// add command.ToolNo
CreateCommandPayload.AddUsint(_command.ToolNo);
// add command.FrameNo
CreateCommandPayload.AddUsint(_command.FrameNo);
// add command.ConnectionMode
CreateCommandPayload.AddUsint(_command.ConnectionMode);
// add command.FixedSensor
CreateCommandPayload.AddByte(_command.FixedSensor);
// add command.SensorFrame[0]
CreateCommandPayload.AddReal(_command.SensorFrame[0]);
// add command.SensorFrame[1]
CreateCommandPayload.AddReal(_command.SensorFrame[1]);
// add command.SensorFrame[2]
CreateCommandPayload.AddReal(_command.SensorFrame[2]);
// add command.SensorFrame[3]
CreateCommandPayload.AddReal(_command.SensorFrame[3]);
// add command.SensorFrame[4]
CreateCommandPayload.AddReal(_command.SensorFrame[4]);
// add command.SensorFrame[5]
CreateCommandPayload.AddReal(_command.SensorFrame[5]);
// add command.CalibrationData
CreateCommandPayload.AddUsint(_command.CalibrationData);
// add command.CalibrationData
CreateCommandPayload.AddUInt(_command.ReferenceType);
// add command.SensorValue[0]
CreateCommandPayload.AddReal(_command.SensorValue[0]);
// add command.SensorValue[1]
CreateCommandPayload.AddReal(_command.SensorValue[1]);
// add command.SensorValue[2]
CreateCommandPayload.AddReal(_command.SensorValue[2]);
// add command.SensorValue[3]
CreateCommandPayload.AddReal(_command.SensorValue[3]);
// add command.SensorValue[4]
CreateCommandPayload.AddReal(_command.SensorValue[4]);
// add command.SensorValue[5]
CreateCommandPayload.AddReal(_command.SensorValue[5]);
// add command.TargetValue[0]
CreateCommandPayload.AddReal(_command.TargetValue[0]);
// add command.TargetValue[1]
CreateCommandPayload.AddReal(_command.TargetValue[1]);
// add command.TargetValue[2]
CreateCommandPayload.AddReal(_command.TargetValue[2]);
// add command.TargetValue[3]
CreateCommandPayload.AddReal(_command.TargetValue[3]);
// add command.TargetValue[4]
CreateCommandPayload.AddReal(_command.TargetValue[4]);
// add command.TargetValue[5]
CreateCommandPayload.AddReal(_command.TargetValue[5]);
// add command.MaxVelocity
CreateCommandPayload.AddUInt(_command.MaxVelocity);
// add command.MaxDeviation[0]
CreateCommandPayload.AddReal(_command.MaxDeviation[0]);
// add command.MaxDeviation[1]
CreateCommandPayload.AddReal(_command.MaxDeviation[1]);
// add command.MaxDeviation[2]
CreateCommandPayload.AddReal(_command.MaxDeviation[2]);
// add command.MaxDeviation[3]
CreateCommandPayload.AddReal(_command.MaxDeviation[3]);
// add command.MaxDeviation[4]
CreateCommandPayload.AddReal(_command.MaxDeviation[4]);
// add command.MaxDeviation[5]
CreateCommandPayload.AddReal(_command.MaxDeviation[5]);
// add command.ErrorReaction
CreateCommandPayload.AddUsint(_command.ErrorReaction);
// add command.ErrorReferenceType
CreateCommandPayload.AddUsint(_command.ErrorReferenceType);
// add command.ErrorVector[0]
CreateCommandPayload.AddReal(_command.ErrorVector[0]);
// add command.ErrorVector[1]
CreateCommandPayload.AddReal(_command.ErrorVector[1]);
// add command.ErrorVector[2]
CreateCommandPayload.AddReal(_command.ErrorVector[2]);
// add command.ErrorVector[3]
CreateCommandPayload.AddReal(_command.ErrorVector[3]);
// add command.ErrorVector[4]
CreateCommandPayload.AddReal(_command.ErrorVector[4]);
// add command.ErrorVector[5]
CreateCommandPayload.AddReal(_command.ErrorVector[5]);
// add command.ErrorToolNo
CreateCommandPayload.AddUsint(_command.ErrorToolNo);
// add command.ErrorFrameNo
CreateCommandPayload.AddUsint(_command.ErrorFrameNo);
// add command.CompliantAxes
CreateCommandPayload.AddByte(_command.CompliantAxes);

// Create logging
CreateCommandPayloadLog(AxesGroup := AxesGroup);
END_METHOD

METHOD INTERNAL CreateCommandPayloadLog 
VAR_IN_OUT
  /// Robot assignment of function
  AxesGroup : AxesGroup; 
END_VAR
// Create log entry for Parameter start
CreateLogMessage      ( Timestamp   := AxesGroup.InternalData.SystemTime,
                        MessageType := MessageType.CMD,
                        Severity    := Severity.DEBUG,
                        MessageCode := 0,
                        MessageText := 'Create command payload with the following parameter(s) :');

// Create log entry for ToolNo
CreateLogMessagePara1 ( Timestamp   := AxesGroup.InternalData.SystemTime,
                        MessageType := MessageType.CMD,
                        Severity    := Severity.DEBUG,
                        MessageCode := 0,
                        MessageText := 'Command.ToolNo = {1}',
                        Para1       :=  USINT_TO_STRING(_command.ToolNo));
                        
// Create log entry for FrameNo
CreateLogMessagePara1 ( Timestamp   := AxesGroup.InternalData.SystemTime,
                        MessageType := MessageType.CMD,
                        Severity    := Severity.DEBUG,
                        MessageCode := 0,
                        MessageText := 'Command.FrameNo = {1}',
                        Para1       :=  USINT_TO_STRING(_command.FrameNo));
                        
// Create log entry for ConnectionMode
CreateLogMessagePara1 ( Timestamp   := AxesGroup.InternalData.SystemTime,
                        MessageType := MessageType.CMD,
                        Severity    := Severity.DEBUG,
                        MessageCode := 0,
                        MessageText := 'Command.ConnectionMode = {1}',
                        Para1       :=  SENSOR_CONNECTION_MODE_TO_STRING(_command.ConnectionMode));

// Create log entry for FixedSensor
CreateLogMessagePara1 ( Timestamp   := AxesGroup.InternalData.SystemTime,
                        MessageType := MessageType.CMD,
                        Severity    := Severity.DEBUG,
                        MessageCode := 0,
                        MessageText := 'Command.FixedSensor = {1}',
                        Para1       :=  BYTE_TO_STRING(_command.FixedSensor));

// Create log entry for SensorFrame[0]
CreateLogMessagePara1 ( Timestamp   := AxesGroup.InternalData.SystemTime,
                        MessageType := MessageType.CMD,
                        Severity    := Severity.DEBUG,
                        MessageCode := 0,
                        MessageText := 'Command.SensorFrame[0] = {1}',
                        Para1       :=  REAL_TO_STRING(_command.SensorFrame[0]));

// Create log entry for SensorFrame[1]
CreateLogMessagePara1 ( Timestamp   := AxesGroup.InternalData.SystemTime,
                        MessageType := MessageType.CMD,
                        Severity    := Severity.DEBUG,
                        MessageCode := 0,
                        MessageText := 'Command.SensorFrame[1] = {1}',
                        Para1       :=  REAL_TO_STRING(_command.SensorFrame[1]));

// Create log entry for SensorFrame[2]
CreateLogMessagePara1 ( Timestamp   := AxesGroup.InternalData.SystemTime,
                        MessageType := MessageType.CMD,
                        Severity    := Severity.DEBUG,
                        MessageCode := 0,
                        MessageText := 'Command.SensorFrame[2] = {1}',
                        Para1       :=  REAL_TO_STRING(_command.SensorFrame[2]));

// Create log entry for SensorFrame[3]
CreateLogMessagePara1 ( Timestamp   := AxesGroup.InternalData.SystemTime,
                        MessageType := MessageType.CMD,
                        Severity    := Severity.DEBUG,
                        MessageCode := 0,
                        MessageText := 'Command.SensorFrame[3] = {1}',
                        Para1       :=  REAL_TO_STRING(_command.SensorFrame[3]));
                                                
// Create log entry for SensorFrame[4]
CreateLogMessagePara1 ( Timestamp   := AxesGroup.InternalData.SystemTime,
                        MessageType := MessageType.CMD,
                        Severity    := Severity.DEBUG,
                        MessageCode := 0,
                        MessageText := 'Command.SensorFrame[4] = {1}',
                        Para1       :=  REAL_TO_STRING(_command.SensorFrame[4]));
                                                
// Create log entry for SensorFrame[5]
CreateLogMessagePara1 ( Timestamp   := AxesGroup.InternalData.SystemTime,
                        MessageType := MessageType.CMD,
                        Severity    := Severity.DEBUG,
                        MessageCode := 0,
                        MessageText := 'Command.SensorFrame[5] = {1}',
                        Para1       :=  REAL_TO_STRING(_command.SensorFrame[5]));

// Create log entry for CalibrationData
CreateLogMessagePara1 ( Timestamp   := AxesGroup.InternalData.SystemTime,
                        MessageType := MessageType.CMD,
                        Severity    := Severity.DEBUG,
                        MessageCode := 0,
                        MessageText := 'Command.CalibrationData = {1}',
                        Para1       :=  USINT_TO_STRING(_command.CalibrationData));
                        
// Create log entry for ReferenceType
CreateLogMessagePara1 ( Timestamp   := AxesGroup.InternalData.SystemTime,
                        MessageType := MessageType.CMD,
                        Severity    := Severity.DEBUG,
                        MessageCode := 0,
                        MessageText := 'Command.ReferenceType = {1}',
                        Para1       :=  REFERENCE_TYPE_TO_STRING(_command.ReferenceType));                        
                                                
// Create log entry for SensorValue[0]
CreateLogMessagePara1 ( Timestamp   := AxesGroup.InternalData.SystemTime,
                        MessageType := MessageType.CMD,
                        Severity    := Severity.DEBUG,
                        MessageCode := 0,
                        MessageText := 'Command.SensorValue[0] = {1}',
                        Para1       :=  REAL_TO_STRING(_command.SensorValue[0]));

// Create log entry for SensorValue[1]
CreateLogMessagePara1 ( Timestamp   := AxesGroup.InternalData.SystemTime,
                        MessageType := MessageType.CMD,
                        Severity    := Severity.DEBUG,
                        MessageCode := 0,
                        MessageText := 'Command.SensorValue[1] = {1}',
                        Para1       :=  REAL_TO_STRING(_command.SensorValue[1]));

// Create log entry for SensorValue[2]
CreateLogMessagePara1 ( Timestamp   := AxesGroup.InternalData.SystemTime,
                        MessageType := MessageType.CMD,
                        Severity    := Severity.DEBUG,
                        MessageCode := 0,
                        MessageText := 'Command.SensorValue[2] = {1}',
                        Para1       :=  REAL_TO_STRING(_command.SensorValue[2]));

// Create log entry for SensorValue[3]
CreateLogMessagePara1 ( Timestamp   := AxesGroup.InternalData.SystemTime,
                        MessageType := MessageType.CMD,
                        Severity    := Severity.DEBUG,
                        MessageCode := 0,
                        MessageText := 'Command.SensorValue[3] = {1}',
                        Para1       :=  REAL_TO_STRING(_command.SensorValue[3]));
                                                
// Create log entry for SensorValue[4]
CreateLogMessagePara1 ( Timestamp   := AxesGroup.InternalData.SystemTime,
                        MessageType := MessageType.CMD,
                        Severity    := Severity.DEBUG,
                        MessageCode := 0,
                        MessageText := 'Command.SensorValue[4] = {1}',
                        Para1       :=  REAL_TO_STRING(_command.SensorValue[4]));
                                                
// Create log entry for SensorValue[5]
CreateLogMessagePara1 ( Timestamp   := AxesGroup.InternalData.SystemTime,
                        MessageType := MessageType.CMD,
                        Severity    := Severity.DEBUG,
                        MessageCode := 0,
                        MessageText := 'Command.SensorValue[5] = {1}',
                        Para1       :=  REAL_TO_STRING(_command.SensorValue[5]));
                                                
// Create log entry for TargetValue[0]
CreateLogMessagePara1 ( Timestamp   := AxesGroup.InternalData.SystemTime,
                        MessageType := MessageType.CMD,
                        Severity    := Severity.DEBUG,
                        MessageCode := 0,
                        MessageText := 'Command.TargetValue[0] = {1}',
                        Para1       :=  REAL_TO_STRING(_command.TargetValue[0]));

// Create log entry for TargetValue[1]
CreateLogMessagePara1 ( Timestamp   := AxesGroup.InternalData.SystemTime,
                        MessageType := MessageType.CMD,
                        Severity    := Severity.DEBUG,
                        MessageCode := 0,
                        MessageText := 'Command.TargetValue[1] = {1}',
                        Para1       :=  REAL_TO_STRING(_command.TargetValue[1]));

// Create log entry for TargetValue[2]
CreateLogMessagePara1 ( Timestamp   := AxesGroup.InternalData.SystemTime,
                        MessageType := MessageType.CMD,
                        Severity    := Severity.DEBUG,
                        MessageCode := 0,
                        MessageText := 'Command.TargetValue[2] = {1}',
                        Para1       :=  REAL_TO_STRING(_command.TargetValue[2]));

// Create log entry for TargetValue[3]
CreateLogMessagePara1 ( Timestamp   := AxesGroup.InternalData.SystemTime,
                        MessageType := MessageType.CMD,
                        Severity    := Severity.DEBUG,
                        MessageCode := 0,
                        MessageText := 'Command.TargetValue[3] = {1}',
                        Para1       :=  REAL_TO_STRING(_command.TargetValue[3]));
                                                
// Create log entry for TargetValue[4]
CreateLogMessagePara1 ( Timestamp   := AxesGroup.InternalData.SystemTime,
                        MessageType := MessageType.CMD,
                        Severity    := Severity.DEBUG,
                        MessageCode := 0,
                        MessageText := 'Command.TargetValue[4] = {1}',
                        Para1       :=  REAL_TO_STRING(_command.TargetValue[4]));
                                                
// Create log entry for TargetValue[5]
CreateLogMessagePara1 ( Timestamp   := AxesGroup.InternalData.SystemTime,
                        MessageType := MessageType.CMD,
                        Severity    := Severity.DEBUG,
                        MessageCode := 0,
                        MessageText := 'Command.TargetValue[5] = {1}',
                        Para1       :=  REAL_TO_STRING(_command.TargetValue[5]));
                                                
// Create log entry for MaxVelocity
CreateLogMessagePara1 ( Timestamp   := AxesGroup.InternalData.SystemTime,
                        MessageType := MessageType.CMD,
                        Severity    := Severity.DEBUG,
                        MessageCode := 0,
                        MessageText := 'Command.MaxVelocity = {1}',
                        Para1       :=  UINT_TO_STRING(_command.MaxVelocity));
                        
// Create log entry for MaxDeviation[0]
CreateLogMessagePara1 ( Timestamp   := AxesGroup.InternalData.SystemTime,
                        MessageType := MessageType.CMD,
                        Severity    := Severity.DEBUG,
                        MessageCode := 0,
                        MessageText := 'Command.MaxDeviation[0] = {1}',
                        Para1       :=  REAL_TO_STRING(_command.MaxDeviation[0]));

// Create log entry for MaxDeviation[1]
CreateLogMessagePara1 ( Timestamp   := AxesGroup.InternalData.SystemTime,
                        MessageType := MessageType.CMD,
                        Severity    := Severity.DEBUG,
                        MessageCode := 0,
                        MessageText := 'Command.MaxDeviation[1] = {1}',
                        Para1       :=  REAL_TO_STRING(_command.MaxDeviation[1]));

// Create log entry for MaxDeviation[2]
CreateLogMessagePara1 ( Timestamp   := AxesGroup.InternalData.SystemTime,
                        MessageType := MessageType.CMD,
                        Severity    := Severity.DEBUG,
                        MessageCode := 0,
                        MessageText := 'Command.MaxDeviation[2] = {1}',
                        Para1       :=  REAL_TO_STRING(_command.MaxDeviation[2]));

// Create log entry for MaxDeviation[3]
CreateLogMessagePara1 ( Timestamp   := AxesGroup.InternalData.SystemTime,
                        MessageType := MessageType.CMD,
                        Severity    := Severity.DEBUG,
                        MessageCode := 0,
                        MessageText := 'Command.MaxDeviation[3] = {1}',
                        Para1       :=  REAL_TO_STRING(_command.MaxDeviation[3]));
                                                
// Create log entry for MaxDeviation[4]
CreateLogMessagePara1 ( Timestamp   := AxesGroup.InternalData.SystemTime,
                        MessageType := MessageType.CMD,
                        Severity    := Severity.DEBUG,
                        MessageCode := 0,
                        MessageText := 'Command.MaxDeviation[4] = {1}',
                        Para1       :=  REAL_TO_STRING(_command.MaxDeviation[4]));
                                                
// Create log entry for MaxDeviation[5]
CreateLogMessagePara1 ( Timestamp   := AxesGroup.InternalData.SystemTime,
                        MessageType := MessageType.CMD,
                        Severity    := Severity.DEBUG,
                        MessageCode := 0,
                        MessageText := 'Command.MaxDeviation[5] = {1}',
                        Para1       :=  REAL_TO_STRING(_command.MaxDeviation[5]));                        
                        
// Create log entry for ErrorReaction
CreateLogMessagePara1 ( Timestamp   := AxesGroup.InternalData.SystemTime,
                        MessageType := MessageType.CMD,
                        Severity    := Severity.DEBUG,
                        MessageCode := 0,
                        MessageText := 'Command.ErrorReaction = {1}',
                        Para1       :=  ERROR_REACTION_TO_STRING(_command.ErrorReaction));    
                        
// Create log entry for ErrorReferenceType
CreateLogMessagePara1 ( Timestamp   := AxesGroup.InternalData.SystemTime,
                        MessageType := MessageType.CMD,
                        Severity    := Severity.DEBUG,
                        MessageCode := 0,
                        MessageText := 'Command.ErrorReferenceType = {1}',
                        Para1       :=  REFERENCE_TYPE_TO_STRING(_command.ErrorReferenceType));     

// Create LOG entry FOR ErrorVector[0]
CreateLogMessagePara1 ( Timestamp   := AxesGroup.InternalData.SystemTime,
                        MessageType := MessageType.CMD,
                        Severity    := Severity.DEBUG,
                        MessageCode := 0,
                        MessageText := 'Command.ErrorVector[0] = {1}',
                        Para1       :=  REAL_TO_STRING(_command.ErrorVector[0]));

// Create log entry for ErrorVector[1]
CreateLogMessagePara1 ( Timestamp   := AxesGroup.InternalData.SystemTime,
                        MessageType := MessageType.CMD,
                        Severity    := Severity.DEBUG,
                        MessageCode := 0,
                        MessageText := 'Command.ErrorVector[1] = {1}',
                        Para1       :=  REAL_TO_STRING(_command.ErrorVector[1]));

// Create log entry for ErrorVector[2]
CreateLogMessagePara1 ( Timestamp   := AxesGroup.InternalData.SystemTime,
                        MessageType := MessageType.CMD,
                        Severity    := Severity.DEBUG,
                        MessageCode := 0,
                        MessageText := 'Command.ErrorVector[2] = {1}',
                        Para1       :=  REAL_TO_STRING(_command.ErrorVector[2]));

// Create log entry for ErrorVector[3]
CreateLogMessagePara1 ( Timestamp   := AxesGroup.InternalData.SystemTime,
                        MessageType := MessageType.CMD,
                        Severity    := Severity.DEBUG,
                        MessageCode := 0,
                        MessageText := 'Command.ErrorVector[3] = {1}',
                        Para1       :=  REAL_TO_STRING(_command.ErrorVector[3]));
                                                
// Create log entry for ErrorVector[4]
CreateLogMessagePara1 ( Timestamp   := AxesGroup.InternalData.SystemTime,
                        MessageType := MessageType.CMD,
                        Severity    := Severity.DEBUG,
                        MessageCode := 0,
                        MessageText := 'Command.ErrorVector[4] = {1}',
                        Para1       :=  REAL_TO_STRING(_command.ErrorVector[4]));
                                                
// Create log entry for ErrorVector[5]
CreateLogMessagePara1 ( Timestamp   := AxesGroup.InternalData.SystemTime,
                        MessageType := MessageType.CMD,
                        Severity    := Severity.DEBUG,
                        MessageCode := 0,
                        MessageText := 'Command.ErrorVector[5] = {1}',
                        Para1       :=  REAL_TO_STRING(_command.ErrorVector[5]));  

// Create log entry for ErrorToolNo
CreateLogMessagePara1 ( Timestamp   := AxesGroup.InternalData.SystemTime,
                        MessageType := MessageType.CMD,
                        Severity    := Severity.DEBUG,
                        MessageCode := 0,
                        MessageText := 'Command.ErrorToolNo = {1}',
                        Para1       :=  USINT_TO_STRING(_command.ErrorToolNo));                                                                                        

// Create log entry for ErrorFrameNo
CreateLogMessagePara1 ( Timestamp   := AxesGroup.InternalData.SystemTime,
                        MessageType := MessageType.CMD,
                        Severity    := Severity.DEBUG,
                        MessageCode := 0,
                        MessageText := 'Command.ErrorFrameNo = {1}',
                        Para1       :=  USINT_TO_STRING(_command.ErrorFrameNo));    

// Create log entry for CompliantAxes
CreateLogMessagePara1 ( Timestamp   := AxesGroup.InternalData.SystemTime,
                        MessageType := MessageType.CMD,
                        Severity    := Severity.DEBUG,
                        MessageCode := 0,
                        MessageText := 'Command.CompliantAxes = {1}',
                        Para1       :=  BYTE_TO_STRING(_command.CompliantAxes));
END_METHOD

METHOD FB_init : BOOL
VAR_INPUT
  /// if TRUE, the retain variables are initialized (warm start / cold start)
  bInitRetains : BOOL; 
  /// if TRUE, the instance afterwards gets moved into the copy code (online change)
  bInCopyCode  : BOOL;  
END_VAR
MyType := 'MC_ForceControlFB';
END_METHOD

METHOD PROTECTED OnCall
VAR_IN_OUT
  /// Robot assignment of function
  AxesGroup : AxesGroup; 
END_VAR
// call base implementation
SUPER^.OnCall(AxesGroup := AxesGroup);

// building rising and falling edges
_enable_R( CLK := Enable);
_enable_F( CLK := Enable);

CASE _stepCmd OF
  
  00:  IF ( _enable_R.Q ) 
       THEN
         // reset the rising edge
        _enable_R();       
         // reset the falling edge
        _enable_F();     

         // Check function is supported and parameter are valid ?
         IF (( CheckFunctionSupported( AxesGroup := AxesGroup )) AND
             ( CheckParameterValid   ( AxesGroup := AxesGroup )))      
         THEN
           // set busy flag
           Busy := TRUE;
           // Reset command outputs
           SysDepMemSet(pDest := ADR(OutCmd), Value := 0, DataLen := SIZEOF(OutCmd));         
           // apply command parameter
          _parCmd := ParCmd;
           // init parameter sequence
          _command.ParSeq := 1;
           // create command data
           CommandData := CreateCommandPayload(AxesGroup := AxesGroup);
           // Add command to active command register
          _uniqueID := AxesGroup.Acyclic.ActiveCommandRegister.AddCmd( pCommandFB := ADR(THIS^ ));     
           // set timeout
           SetTimeout(PT := _timeoutCmd, rTimer := _timerCmd);
           // inc step counter
          _stepCmd := _stepCmd + 1; 
         END_IF   
       END_IF
     

  01:  // Wait for responce received
       IF ( _responseReceived )
       THEN
         // reset response received flag
        _responseReceived := FALSE;

         CASE  _response.State 
         OF
           CmdMessageState.BUFFERED    : CommandBuffered    := TRUE;
           CmdMessageState.ACTIVE      : ParameterAccepted  := TRUE;
                                         Valid              := TRUE;
           CmdMessageState.ERROR       : Error              := TRUE;
         END_CASE
         
         // Done, Aborted or Error ?
         IF (_response.State >= CmdMessageState.DONE )
         THEN
           // Update results
           OutCmd.ForceStatus.ForceControlEnabled         := _response.ForceStatus.0;
           OutCmd.ForceStatus.ForceLimitEnabled           := _response.ForceStatus.1;
           OutCmd.ForceStatus.ApplyingForce               := _response.ForceStatus.2;
           OutCmd.ForceStatus.MaxDeviationReached         := _response.ForceStatus.3;
           OutCmd.ForceStatus.SpecifiedForceTorqueReached := _response.ForceStatus.4;
           OutCmd.ForceStatus.SpecifiedForceLimitReached  := _response.ForceStatus.5;
           OutCmd.ForceStatus.Bit06                       := _response.ForceStatus.6;
           OutCmd.ForceStatus.Bit07                       := _response.ForceStatus.7;  
           // set timeout
           SetTimeout(PT := _timeoutCmd, rTimer := _timerCmd);
           // inc step counter
          _stepCmd := _stepCmd + 1;
         END_IF
 
       END_IF


  02: IF (NOT Enable)
      THEN
        Reset();
	    END_IF
ELSE
  // invalid step
  ErrorID := RobotLibraryEvents.ERR_INVALID_STEP;
END_CASE



// Reset FB
IF (( _enable_R.Q ) OR
    ( _enable_F.Q ))
THEN
 _uniqueId           := 0;
 _stepCmd            := 0;
  Valid              := FALSE;
  Busy               := FALSE;
  CommandBuffered    := FALSE;
  Error              := FALSE;
  ErrorID            := 0;
  WarningID          := 0;
  InfoID             := 0;  
END_IF
END_METHOD

METHOD INTERNAL ParseResponsePayload : DINT
VAR_INPUT
  /// Response data
  ResponseData : RobotLibraryRecvDataFB;
  /// Timestamp
  Timestamp    : SystemTime;  
END_VAR
// Table 6-720: Received CMD payload (RC to PLC) of "ForceControl"
// --------------------------
// Header
// --------------------------
// Byte 00 : USINT      - ParSeq | State     
// Byte 01 : SINT       - AlarmMessageSeverity    
// Byte 02 : UINT       - AlarmMessageCode HB
// Byte 03 :            - AlarmMessageCode LB
// --------------------------
// Datablock
// --------------------------
// Byte 04 : USINT      - ForceStatus 
// --------------------------
// call base implementation to parse the header from payload buffer
ResponseData.PayloadPtr := SUPER^.ParseResponsePayload(ResponseData := ResponseData, Timestamp := Timestamp);

// copy parsed header to response
_response.ParSeq                := _rspHeader.ParSeq;
_response.State                 := _rspHeader.State;
_response.AlarmMessageSeverity  := _rspHeader.AlarmMessageSeverity;
_response.AlarmMessageCode      := _rspHeader.AlarmMessageCode;

// Get Response.ForceStatus
_response.ForceStatus := ResponseData.GetByte();

// Create logging
ParseResponsePayloadLog(ResponseData := ResponseData, Timestamp := Timestamp);
END_METHOD

METHOD INTERNAL ParseResponsePayloadLog
VAR_INPUT
  /// Response data
  ResponseData : RobotLibraryRecvDataFB;
  /// Timestamp
  Timestamp    : SystemTime;  
END_VAR
// Create log entry for Parameter start
CreateLogMessage      ( Timestamp   := Timestamp,
                        MessageType := MessageType.CMD,
                        Severity    := Severity.DEBUG,
                        MessageCode := 0,
                        MessageText := 'Parsed the following parameter(s) from response data:');
                        
// Create log entry for ForceStatus
CreateLogMessagePara1 ( Timestamp   := Timestamp,
                        MessageType := MessageType.CMD,
                        Severity    := Severity.DEBUG,
                        MessageCode := 0,
                        MessageText := 'Response.ForceStatus = {1}',
                        Para1       :=  BYTE_TO_STRING(_response.ForceStatus));
END_METHOD

METHOD PROTECTED Reset : DINT
VAR_INPUT
END_VAR
Reset := SUPER^.Reset();

Valid              := FALSE;
Busy               := FALSE;
CommandBuffered    := FALSE;
ParameterAccepted  := FALSE;
END_METHOD

END_FUNCTION_BLOCK

// Library/POUs/ForceControl/MC_ForceLimit/MC_ForceLimitFB
/// Commands specified reaction from RA when defined force/torque detected
FUNCTION_BLOCK MC_ForceLimitFB EXTENDS RobotLibraryBaseFB
// ------------------------------------------------------------------------- 
//  SRCI Robot Library                                                
// ------------------------------------------------------------------------- 
//                                                                           
//  Object:      ForceLimitFB                                       
//  Author:      Thorsten Brach                                                
//  Date:        2024-06-01
//
//  Description:                                              
//   
//                                                                           
//  Copyright: 
//    (C) 2024 Thorsten Brach. All rights reserved                                                                                                                                            
//             Licensed under the LGPL-3.0 license.
//                                                                           
//  Disclaimer:                                                                           
//    This project is provided without any guarantee and can be used for   
//    private and commercial purposes. Any use is at the user’s 
//    own risk and responsibility.
//
// -------------------------------------------------------------------------
VAR_INPUT
  /// Set TRUE to activate force limiting
  Enable            : BOOL;
  /// Command parameter 
  ParCmd            : ForceLimitParCmd;   
END_VAR

VAR_OUTPUT
  /// TRUE, while the following outputs return valid values
  Valid             : BOOL;
  /// FB is being processed
  Busy              : BOOL;
  /// Command is transferred and confirmed by the RC
  CommandBuffered   : BOOL;
  /// Receiving of input parameter values has been acknowledged by RC
  ParameterAccepted : BOOL;
  /// Command output 
  OutCmd            : ForceLimitOutCmd;      
END_VAR


VAR
  /// internal copy of command parameter 
 _parCmd            : ForceLimitParCmd;
  /// command data to send
 _command           : ForceLimitSendData;
  /// response data received
 _response          : ForceLimitRecvData;      
  /// Rising edge for enable
 _enable_R          : R_TRIG;
  /// Falling edge for enable
 _enable_F          : F_TRIG;  
END_VAR

SUPER^(AxesGroup := AxesGroup);

METHOD PROTECTED CheckFunctionSupported : BOOL
VAR_IN_OUT
  /// Robot assignment of function
  AxesGroup : AxesGroup; 
END_VAR
CheckFunctionSupported := AxesGroup.InternalData.RCSupportedFunctions.ForceLimit;

IF ( NOT CheckFunctionSupported )
THEN
  // call base implementation for set error and create log entry
  SUPER^.CheckFunctionSupported(AxesGroup := AxesGroup);
END_IF
END_METHOD

METHOD PROTECTED CheckParameterChanged : BOOL
VAR_IN_OUT
  /// Robot assignment of function
  AxesGroup    : AxesGroup; 
END_VAR
// Check ParCmd Size is > 0, because MemCmp does not work correctly with size = 0
IF (SIZEOF(ParCmd) = 0) 
THEN 
  RETURN;
END_IF

// compare memory 
_parameterChanged := ( SysDepMemCmp(pData1 := ADR(ParCmd), pData2 := ADR(_parCmd), DataLen := SIZEOF(ParCmd)) <> RobotLibraryConstants.OK );

// check parameter valid ?
_parameterValid   := CheckParameterValid( AxesGroup := AxesGroup );

IF ((  _parameterChanged        )  AND 
    (  _parameterValid          )) OR
    (  _parameterUpdateInternal )  
THEN  
  // reset internal flag for send parameter update
 _parameterUpdateInternal := FALSE;
  // update internal copy of parameters 
 _parCmd := ParCmd;
  // inc parameter sequence
 _command.ParSeq := _command.ParSeq + 1;
  // update command data  
  CommandData := CreateCommandPayload(AxesGroup := AxesGroup); // ( Access via reference to rCommandFB in ACR )
  // notify active command register 
  AxesGroup.Acyclic.ActiveCommandRegister.NotifyParameterChanged := _uniqueID;
  // Reset parameter accepted flag
  ParameterAccepted := FALSE;  
END_IF
END_METHOD

METHOD INTERNAL CreateCommandPayload : RobotLibrarySendDataFB
VAR_IN_OUT
  /// Robot assignment of function
  AxesGroup : AxesGroup; 
END_VAR
// Table 6-727: Sent CMD payload (PLC to RC) of "ForceLimit"
// --------------------------
// Header
// --------------------------
// Byte 00 : UINT       - Type HB     
// Byte 01 :            - Type LB    
// Byte 02 : USINT      - Reserve | ExecutionMode
// Byte 03 : USINT      - ParSeq  | Priority
// --------------------------
// Datablock
// --------------------------
// Byte 004 : SINT       - EmitterID[0] 
// Byte 005 : SINT       - EmitterID[1] 
// Byte 006 : SINT       - EmitterID[2] 
// Byte 007 : SINT       - EmitterID[3]
// Byte 008 : SINT       - ListenerID
// Byte 009 : BYTE       - Reserve
// Byte 010 : USINT      - ToolNo
// Byte 011 : USINT      - FrameNo
// Byte 012 : USINT      - ConnectionMode
// Byte 013 : BOOL       - FixedSensor
// Byte 014 : REAL       - SensorFrame[0] HW HB
// Byte 015 :            - SensorFrame[0] HW LB
// Byte 016 :            - SensorFrame[0] LW HB
// Byte 017 :            - SensorFrame[0] LW LB
// Byte 018 : REAL       - SensorFrame[1] HW HB
// Byte 019 :            - SensorFrame[1] HW LB
// Byte 020 :            - SensorFrame[1] LW HB
// Byte 021 :            - SensorFrame[1] LW LB
// Byte 022 : REAL       - SensorFrame[2] HW HB
// Byte 023 :            - SensorFrame[2] HW LB
// Byte 024 :            - SensorFrame[2] LW HB
// Byte 025 :            - SensorFrame[2] LW LB
// Byte 026 : REAL       - SensorFrame[3] HW HB
// Byte 027 :            - SensorFrame[3] HW LB
// Byte 028 :            - SensorFrame[3] LW HB
// Byte 029 :            - SensorFrame[3] LW LB
// Byte 030 : REAL       - SensorFrame[4] HW HB
// Byte 031 :            - SensorFrame[4] HW LB
// Byte 032 :            - SensorFrame[4] LW HB
// Byte 033 :            - SensorFrame[4] LW LB
// Byte 034 : REAL       - SensorFrame[5] HW HB
// Byte 035 :            - SensorFrame[5] HW LB
// Byte 036 :            - SensorFrame[5] LW HB
// Byte 037 :            - SensorFrame[5] LW LB
// Byte 038 : USINT      - CalibrationData
// Byte 039 : USINT      - ReferenceType
// Byte 040 : REAL       - SensorValue[0] HW HB
// Byte 041 :            - SensorValue[0] HW LB
// Byte 042 :            - SensorValue[0] LW HB
// Byte 043 :            - SensorValue[0] LW LB
// Byte 044 : REAL       - SensorValue[1] HW HB
// Byte 045 :            - SensorValue[1] HW LB
// Byte 046 :            - SensorValue[1] LW HB
// Byte 047 :            - SensorValue[1] LW LB
// Byte 048 : REAL       - SensorValue[2] HW HB
// Byte 049 :            - SensorValue[2] HW LB
// Byte 050 :            - SensorValue[2] LW HB
// Byte 051 :            - SensorValue[2] LW LB
// Byte 052 : REAL       - SensorValue[3] HW HB
// Byte 053 :            - SensorValue[3] HW LB
// Byte 054 :            - SensorValue[3] LW HB
// Byte 055 :            - SensorValue[3] LW LB
// Byte 056 : REAL       - SensorValue[4] HW HB
// Byte 057 :            - SensorValue[4] HW LB
// Byte 058 :            - SensorValue[4] LW HB
// Byte 059 :            - SensorValue[4] LW LB
// Byte 060 : REAL       - SensorValue[5] HW HB
// Byte 061 :            - SensorValue[5] HW LB
// Byte 062 :            - SensorValue[5] LW HB
// Byte 063 :            - SensorValue[5] LW LB
// Byte 064 : REAL       - Limit[0] HW HB
// Byte 065 :            - Limit[0] HW LB
// Byte 066 :            - Limit[0] LW HB
// Byte 067 :            - Limit[0] LW LB
// Byte 068 : REAL       - Limit[1] HW HB
// Byte 069 :            - Limit[1] HW LB
// Byte 070 :            - Limit[1] LW HB
// Byte 071 :            - Limit[1] LW LB
// Byte 072 : REAL       - Limit[2] HW HB
// Byte 073 :            - Limit[2] HW LB
// Byte 074 :            - Limit[2] LW HB
// Byte 075 :            - Limit[2] LW LB
// Byte 076 : REAL       - Limit[3] HW HB
// Byte 077 :            - Limit[3] HW LB
// Byte 078 :            - Limit[3] LW HB
// Byte 079 :            - Limit[3] LW LB
// Byte 080 : REAL       - Limit[4] HW HB
// Byte 081 :            - Limit[4] HW LB
// Byte 082 :            - Limit[4] LW HB
// Byte 083 :            - Limit[4] LW LB
// Byte 084 : REAL       - Limit[5] HW HB
// Byte 085 :            - Limit[5] HW LB
// Byte 086 :            - Limit[5] LW HB
// Byte 087 :            - Limit[5] LW LB


// --------------------------
// set command parameter 
_command.CmdTyp          :=  CmdType.ForceLimit;
_command.ExecMode        :=  ExecMode;
_command.ParSeq          := _command.ParSeq;
_command.Priority        :=  Priority;
_command.EmitterID[0]    := _parCmd.EmitterID;
_command.ListenerID      :=  0; {warning 'ToDo'} 
_command.Reserve         :=  0; 
_command.ToolNo          := _parCmd.ToolNo;
_command.FrameNo         := _parCmd.FrameNo;
_command.ConnectionMode  := _parCmd.ConnectionMode;
_command.FixedSensor.0   := _parCmd.FixedSensor;
_command.SensorFrame     := _parCmd.SensorFrame;
_command.CalibrationData := _parCmd.CalibrationData;
_command.ReferenceType   := _parCmd.ReferenceType;
_command.SensorValue     := _parCmd.SensorValue;
_command.ForceLimit      := _parCmd.ForceLimit;  



// copy command data to header
_cmdHeader := _command;
// call base implementation to copy header to payload buffer
CreateCommandPayload := SUPER^.CreateCommandPayload(AxesGroup := AxesGroup);


// add command.EmitterID[0]
CreateCommandPayload.AddSint(_command.EmitterID[0]);
// add command.EmitterID[1]
CreateCommandPayload.AddSint(_command.EmitterID[1]);
// add command.EmitterID[2]
CreateCommandPayload.AddSint(_command.EmitterID[2]);
// add command.EmitterID[3]
CreateCommandPayload.AddSint(_command.EmitterID[3]);
// add command.ListenerID
CreateCommandPayload.AddSint(_command.ListenerID);
// add command.Reserve
CreateCommandPayload.AddByte(_command.Reserve);
// add command.ToolNo
CreateCommandPayload.AddUsint(_command.ToolNo);
// add command.FrameNo
CreateCommandPayload.AddUsint(_command.FrameNo);
// add command.ConnectionMode
CreateCommandPayload.AddUsint(_command.ConnectionMode);
// add command.FixedSensor
CreateCommandPayload.AddByte(_command.FixedSensor);
// add command.SensorFrame[0]
CreateCommandPayload.AddReal(_command.SensorFrame[0]);
// add command.SensorFrame[1]
CreateCommandPayload.AddReal(_command.SensorFrame[1]);
// add command.SensorFrame[2]
CreateCommandPayload.AddReal(_command.SensorFrame[2]);
// add command.SensorFrame[3]
CreateCommandPayload.AddReal(_command.SensorFrame[3]);
// add command.SensorFrame[4]
CreateCommandPayload.AddReal(_command.SensorFrame[4]);
// add command.SensorFrame[5]
CreateCommandPayload.AddReal(_command.SensorFrame[5]);
// add command.CalibrationData
CreateCommandPayload.AddUsint(_command.CalibrationData);
// add command.ReferenceType
CreateCommandPayload.AddUsint(_command.ReferenceType);
// add command.SensorValue[0]
CreateCommandPayload.AddReal(_command.SensorValue[0]);
// add command.SensorValue[1]
CreateCommandPayload.AddReal(_command.SensorValue[1]);
// add command.SensorValue[2]
CreateCommandPayload.AddReal(_command.SensorValue[2]);
// add command.SensorValue[3]
CreateCommandPayload.AddReal(_command.SensorValue[3]);
// add command.SensorValue[4]
CreateCommandPayload.AddReal(_command.SensorValue[4]);
// add command.SensorValue[5]
CreateCommandPayload.AddReal(_command.SensorValue[5]);

// add command.ForceLimit[0]
CreateCommandPayload.AddReal(_command.ForceLimit[0]);
// add command.ForceLimit[1]
CreateCommandPayload.AddReal(_command.ForceLimit[1]);
// add command.ForceLimit[2]
CreateCommandPayload.AddReal(_command.ForceLimit[2]);
// add command.ForceLimit[3]
CreateCommandPayload.AddReal(_command.ForceLimit[3]);
// add command.ForceLimit[4]
CreateCommandPayload.AddReal(_command.ForceLimit[4]);
// add command.ForceLimit[5]
CreateCommandPayload.AddReal(_command.ForceLimit[5]);

// Create logging
CreateCommandPayloadLog(AxesGroup := AxesGroup);
END_METHOD

METHOD INTERNAL CreateCommandPayloadLog 
VAR_IN_OUT
  /// Robot assignment of function
  AxesGroup : AxesGroup; 
END_VAR
VAR 
  /// internal index for loops
 _idx : DINT;
END_VAR
// Create log entry for Parameter start
CreateLogMessage      ( Timestamp   := AxesGroup.InternalData.SystemTime,
                        MessageType := MessageType.CMD,
                        Severity    := Severity.DEBUG,
                        MessageCode := 0,
                        MessageText := 'Create command payload with the following parameter(s) :');

// Create log entry for EmitterID[0]
CreateLogMessagePara1 ( Timestamp   := AxesGroup.InternalData.SystemTime,
                        MessageType := MessageType.CMD,
                        Severity    := Severity.DEBUG,
                        MessageCode := 0,
                        MessageText := 'Command.EmitterID[0] = {1}',
                        Para1       :=  SINT_TO_STRING(_command.EmitterID[0]));

// Create log entry for EmitterID[x]
FOR _idx := 0 TO 3
DO
  CreateLogMessagePara2 ( Timestamp   := AxesGroup.InternalData.SystemTime,
                          MessageType := MessageType.CMD,
                          Severity    := Severity.DEBUG,
                          MessageCode := 0,
                          MessageText := 'Command.EmitterID[{2}] = {1}',
                          Para1       :=  SINT_TO_STRING(_command.EmitterID[_idx]),
                          Para2       :=  DINT_TO_STRING(_idx));
END_FOR

// Create log entry for ListenerID
CreateLogMessagePara1 ( Timestamp   := AxesGroup.InternalData.SystemTime,
                        MessageType := MessageType.CMD,
                        Severity    := Severity.DEBUG,
                        MessageCode := 0,
                        MessageText := 'Command.ListenerID = {1}',
                        Para1       :=  SINT_TO_STRING(_command.ListenerID));
                        
// Create log entry for Reserve
CreateLogMessagePara1 ( Timestamp   := AxesGroup.InternalData.SystemTime,
                        MessageType := MessageType.CMD,
                        Severity    := Severity.DEBUG,
                        MessageCode := 0,
                        MessageText := 'Command.Reserve = {1}',
                        Para1       :=  BYTE_TO_STRING(_command.Reserve));

// Create log entry for ToolNo
CreateLogMessagePara1 ( Timestamp   := AxesGroup.InternalData.SystemTime,
                        MessageType := MessageType.CMD,
                        Severity    := Severity.DEBUG,
                        MessageCode := 0,
                        MessageText := 'Command.ToolNo = {1}',
                        Para1       :=  USINT_TO_STRING(_command.ToolNo));
                        
// Create log entry for FrameNo
CreateLogMessagePara1 ( Timestamp   := AxesGroup.InternalData.SystemTime,
                        MessageType := MessageType.CMD,
                        Severity    := Severity.DEBUG,
                        MessageCode := 0,
                        MessageText := 'Command.FrameNo = {1}',
                        Para1       :=  USINT_TO_STRING(_command.FrameNo));
                        
// Create log entry for ConnectionMode
CreateLogMessagePara1 ( Timestamp   := AxesGroup.InternalData.SystemTime,
                        MessageType := MessageType.CMD,
                        Severity    := Severity.DEBUG,
                        MessageCode := 0,
                        MessageText := 'Command.ConnectionMode = {1}',
                        Para1       :=  SENSOR_CONNECTION_MODE_TO_STRING(_command.ConnectionMode));

// Create log entry for FixedSensor
CreateLogMessagePara1 ( Timestamp   := AxesGroup.InternalData.SystemTime,
                        MessageType := MessageType.CMD,
                        Severity    := Severity.DEBUG,
                        MessageCode := 0,
                        MessageText := 'Command.FixedSensor = {1}',
                        Para1       :=  BYTE_TO_STRING(_command.FixedSensor));

// Create log entry for SensorFrame[0]
CreateLogMessagePara1 ( Timestamp   := AxesGroup.InternalData.SystemTime,
                        MessageType := MessageType.CMD,
                        Severity    := Severity.DEBUG,
                        MessageCode := 0,
                        MessageText := 'Command.SensorFrame[0] = {1}',
                        Para1       :=  REAL_TO_STRING(_command.SensorFrame[0]));

// Create log entry for SensorFrame[1]
CreateLogMessagePara1 ( Timestamp   := AxesGroup.InternalData.SystemTime,
                        MessageType := MessageType.CMD,
                        Severity    := Severity.DEBUG,
                        MessageCode := 0,
                        MessageText := 'Command.SensorFrame[1] = {1}',
                        Para1       :=  REAL_TO_STRING(_command.SensorFrame[1]));

// Create log entry for SensorFrame[2]
CreateLogMessagePara1 ( Timestamp   := AxesGroup.InternalData.SystemTime,
                        MessageType := MessageType.CMD,
                        Severity    := Severity.DEBUG,
                        MessageCode := 0,
                        MessageText := 'Command.SensorFrame[2] = {1}',
                        Para1       :=  REAL_TO_STRING(_command.SensorFrame[2]));

// Create log entry for SensorFrame[3]
CreateLogMessagePara1 ( Timestamp   := AxesGroup.InternalData.SystemTime,
                        MessageType := MessageType.CMD,
                        Severity    := Severity.DEBUG,
                        MessageCode := 0,
                        MessageText := 'Command.SensorFrame[3] = {1}',
                        Para1       :=  REAL_TO_STRING(_command.SensorFrame[3]));
                                                
// Create log entry for SensorFrame[4]
CreateLogMessagePara1 ( Timestamp   := AxesGroup.InternalData.SystemTime,
                        MessageType := MessageType.CMD,
                        Severity    := Severity.DEBUG,
                        MessageCode := 0,
                        MessageText := 'Command.SensorFrame[4] = {1}',
                        Para1       :=  REAL_TO_STRING(_command.SensorFrame[4]));
                                                
// Create log entry for SensorFrame[5]
CreateLogMessagePara1 ( Timestamp   := AxesGroup.InternalData.SystemTime,
                        MessageType := MessageType.CMD,
                        Severity    := Severity.DEBUG,
                        MessageCode := 0,
                        MessageText := 'Command.SensorFrame[5] = {1}',
                        Para1       :=  REAL_TO_STRING(_command.SensorFrame[5]));

// Create log entry for CalibrationData
CreateLogMessagePara1 ( Timestamp   := AxesGroup.InternalData.SystemTime,
                        MessageType := MessageType.CMD,
                        Severity    := Severity.DEBUG,
                        MessageCode := 0,
                        MessageText := 'Command.CalibrationData = {1}',
                        Para1       :=  USINT_TO_STRING(_command.CalibrationData));
                        
// Create log entry for ReferenceType
CreateLogMessagePara1 ( Timestamp   := AxesGroup.InternalData.SystemTime,
                        MessageType := MessageType.CMD,
                        Severity    := Severity.DEBUG,
                        MessageCode := 0,
                        MessageText := 'Command.ReferenceType = {1}',
                        Para1       :=  REFERENCE_TYPE_TO_STRING(_command.ReferenceType));                        
                                                
// Create log entry for SensorValue[0]
CreateLogMessagePara1 ( Timestamp   := AxesGroup.InternalData.SystemTime,
                        MessageType := MessageType.CMD,
                        Severity    := Severity.DEBUG,
                        MessageCode := 0,
                        MessageText := 'Command.SensorValue[0] = {1}',
                        Para1       :=  REAL_TO_STRING(_command.SensorValue[0]));

// Create log entry for SensorValue[1]
CreateLogMessagePara1 ( Timestamp   := AxesGroup.InternalData.SystemTime,
                        MessageType := MessageType.CMD,
                        Severity    := Severity.DEBUG,
                        MessageCode := 0,
                        MessageText := 'Command.SensorValue[1] = {1}',
                        Para1       :=  REAL_TO_STRING(_command.SensorValue[1]));

// Create log entry for SensorValue[2]
CreateLogMessagePara1 ( Timestamp   := AxesGroup.InternalData.SystemTime,
                        MessageType := MessageType.CMD,
                        Severity    := Severity.DEBUG,
                        MessageCode := 0,
                        MessageText := 'Command.SensorValue[2] = {1}',
                        Para1       :=  REAL_TO_STRING(_command.SensorValue[2]));

// Create log entry for SensorValue[3]
CreateLogMessagePara1 ( Timestamp   := AxesGroup.InternalData.SystemTime,
                        MessageType := MessageType.CMD,
                        Severity    := Severity.DEBUG,
                        MessageCode := 0,
                        MessageText := 'Command.SensorValue[3] = {1}',
                        Para1       :=  REAL_TO_STRING(_command.SensorValue[3]));
                                                
// Create log entry for SensorValue[4]
CreateLogMessagePara1 ( Timestamp   := AxesGroup.InternalData.SystemTime,
                        MessageType := MessageType.CMD,
                        Severity    := Severity.DEBUG,
                        MessageCode := 0,
                        MessageText := 'Command.SensorValue[4] = {1}',
                        Para1       :=  REAL_TO_STRING(_command.SensorValue[4]));
                                                
// Create log entry for SensorValue[5]
CreateLogMessagePara1 ( Timestamp   := AxesGroup.InternalData.SystemTime,
                        MessageType := MessageType.CMD,
                        Severity    := Severity.DEBUG,
                        MessageCode := 0,
                        MessageText := 'Command.SensorValue[5] = {1}',
                        Para1       :=  REAL_TO_STRING(_command.SensorValue[5]));
                                                
// Create log entry for ForceLimit[0]
CreateLogMessagePara1 ( Timestamp   := AxesGroup.InternalData.SystemTime,
                        MessageType := MessageType.CMD,
                        Severity    := Severity.DEBUG,
                        MessageCode := 0,
                        MessageText := 'Command.ForceLimit[0] = {1}',
                        Para1       :=  REAL_TO_STRING(_command.ForceLimit[0]));

// Create log entry for ForceLimit[1]
CreateLogMessagePara1 ( Timestamp   := AxesGroup.InternalData.SystemTime,
                        MessageType := MessageType.CMD,
                        Severity    := Severity.DEBUG,
                        MessageCode := 0,
                        MessageText := 'Command.ForceLimit[1] = {1}',
                        Para1       :=  REAL_TO_STRING(_command.ForceLimit[1]));

// Create log entry for ForceLimit[2]
CreateLogMessagePara1 ( Timestamp   := AxesGroup.InternalData.SystemTime,
                        MessageType := MessageType.CMD,
                        Severity    := Severity.DEBUG,
                        MessageCode := 0,
                        MessageText := 'Command.ForceLimit[2] = {1}',
                        Para1       :=  REAL_TO_STRING(_command.ForceLimit[2]));

// Create log entry for ForceLimit[3]
CreateLogMessagePara1 ( Timestamp   := AxesGroup.InternalData.SystemTime,
                        MessageType := MessageType.CMD,
                        Severity    := Severity.DEBUG,
                        MessageCode := 0,
                        MessageText := 'Command.ForceLimit[3] = {1}',
                        Para1       :=  REAL_TO_STRING(_command.ForceLimit[3]));
                                                
// Create log entry for ForceLimit[4]
CreateLogMessagePara1 ( Timestamp   := AxesGroup.InternalData.SystemTime,
                        MessageType := MessageType.CMD,
                        Severity    := Severity.DEBUG,
                        MessageCode := 0,
                        MessageText := 'Command.ForceLimit[4] = {1}',
                        Para1       :=  REAL_TO_STRING(_command.ForceLimit[4]));
                                                
// Create log entry for ForceLimit[5]
CreateLogMessagePara1 ( Timestamp   := AxesGroup.InternalData.SystemTime,
                        MessageType := MessageType.CMD,
                        Severity    := Severity.DEBUG,
                        MessageCode := 0,
                        MessageText := 'Command.ForceLimit[5] = {1}',
                        Para1       :=  REAL_TO_STRING(_command.ForceLimit[5]));
END_METHOD

METHOD FB_init : BOOL
VAR_INPUT
  /// if TRUE, the retain variables are initialized (warm start / cold start)
  bInitRetains : BOOL; 
  /// if TRUE, the instance afterwards gets moved into the copy code (online change)
  bInCopyCode  : BOOL;  
END_VAR
MyType := 'MC_ForceLimitFB';
END_METHOD

METHOD PROTECTED OnCall
VAR_IN_OUT
  /// Robot assignment of function
  AxesGroup : AxesGroup; 
END_VAR
// call base implementation
SUPER^.OnCall(AxesGroup := AxesGroup);

// building rising and falling edges
_enable_R( CLK := Enable);
_enable_F( CLK := Enable);

CASE _stepCmd OF
  
  00:  IF ( _enable_R.Q ) 
       THEN
         // reset the rising edge
        _enable_R();       
         // reset the falling edge
        _enable_F();       

         // Check function is supported and parameter are valid ?
         IF (( CheckFunctionSupported( AxesGroup := AxesGroup )) AND
             ( CheckParameterValid   ( AxesGroup := AxesGroup )))      
         THEN
           // set busy flag
           Busy := TRUE;
           // Reset command outputs
           SysDepMemSet(pDest := ADR(OutCmd), Value := 0, DataLen := SIZEOF(OutCmd));         
           // apply command parameter
          _parCmd := ParCmd;
           // init parameter sequence
          _command.ParSeq := 1;
           // create command data
           CommandData := CreateCommandPayload(AxesGroup := AxesGroup);
           // Add command to active command register
          _uniqueID := AxesGroup.Acyclic.ActiveCommandRegister.AddCmd( pCommandFB := ADR(THIS^ ));     
           // set timeout
           SetTimeout(PT := _timeoutCmd, rTimer := _timerCmd);
           // inc step counter
          _stepCmd := _stepCmd + 1;
         END_IF 
       END_IF
     

  01:  // Wait for responce received
       IF ( _responseReceived )
       THEN
         // reset response received flag
        _responseReceived := FALSE;

         CASE  _response.State 
         OF
           CmdMessageState.BUFFERED    : CommandBuffered    := TRUE;
           CmdMessageState.ACTIVE      : ParameterAccepted  := TRUE;
                                         Valid              := TRUE;
           CmdMessageState.ERROR       : Error              := TRUE;
         END_CASE
         // Done, Aborted or Error ?
         IF (_response.State >= CmdMessageState.DONE )
         THEN         
           // Update results
           OutCmd.ForceStatus.ForceControlEnabled         := _response.ForceStatus.0;
           OutCmd.ForceStatus.ForceLimitEnabled           := _response.ForceStatus.1;
           OutCmd.ForceStatus.ApplyingForce               := _response.ForceStatus.2;
           OutCmd.ForceStatus.MaxDeviationReached         := _response.ForceStatus.3;
           OutCmd.ForceStatus.SpecifiedForceTorqueReached := _response.ForceStatus.4;
           OutCmd.ForceStatus.SpecifiedForceLimitReached  := _response.ForceStatus.5;
           OutCmd.ForceStatus.Bit06                       := _response.ForceStatus.6;
           OutCmd.ForceStatus.Bit07                       := _response.ForceStatus.7;  
           OutCmd.FollowID                                := _response.OriginID; {warning 'ToDo'}
           // set timeout
           SetTimeout(PT := _timeoutCmd, rTimer := _timerCmd);
           // inc step counter
          _stepCmd := _stepCmd + 1;
         END_IF
 
       END_IF


  02: IF (NOT Enable)
      THEN
        Reset();
	    END_IF

ELSE
  // invalid step
  ErrorID := RobotLibraryEvents.ERR_INVALID_STEP;
END_CASE



// Reset FB
IF (( _enable_R.Q ) OR
    ( _enable_F.Q ))
THEN
 _uniqueId           := 0;
 _stepCmd            := 0;
  Valid              := FALSE;
  Busy               := FALSE;
  CommandBuffered    := FALSE;
  Error              := FALSE;
  ErrorID            := 0;
  WarningID          := 0;
  InfoID             := 0;  
END_IF
END_METHOD

METHOD INTERNAL ParseResponsePayload : DINT
VAR_INPUT
  /// Response data
  ResponseData : RobotLibraryRecvDataFB;
  /// Timestamp
  Timestamp    : SystemTime;  
END_VAR
// Table 6-728: Received CMD payload (RC to PLC) of "ForceLimit"
// --------------------------
// Header
// --------------------------
// Byte 00 : USINT      - ParSeq | State     
// Byte 01 : SINT       - AlarmMessageSeverity    
// Byte 02 : UINT       - AlarmMessageCode HB
// Byte 03 :            - AlarmMessageCode LB
// --------------------------
// Datablock
// --------------------------
// Byte 04 : USINT      - InvocationCounter 
// Byte 05 : USINT      - Reserved 
// Byte 06 : INT        - OriginID LW HB
// Byte 07 :            - OriginID LW LB 
// Byte 08 : BYTE       - ForceStatus 
// --------------------------
// call base implementation to parse the header from payload buffer
ResponseData.PayloadPtr := SUPER^.ParseResponsePayload(ResponseData := ResponseData, Timestamp := Timestamp);

// copy parsed header to response
_response.ParSeq                := _rspHeader.ParSeq;
_response.State                 := _rspHeader.State;
_response.AlarmMessageSeverity  := _rspHeader.AlarmMessageSeverity;
_response.AlarmMessageCode      := _rspHeader.AlarmMessageCode;

// Get Response.InvocationCounter
_response.InvocationCounter := ResponseData.GetUsint();
// Get Response.Reserved
_response.Reserved := ResponseData.GetSint();
// Get Response.OriginID
_response.OriginID := ResponseData.GetInt();
// Get Response.ForceStatus
_response.ForceStatus := ResponseData.GetByte();

// Create logging
ParseResponsePayloadLog(ResponseData := ResponseData, Timestamp := Timestamp);
END_METHOD

METHOD INTERNAL ParseResponsePayloadLog
VAR_INPUT
  /// Response data
  ResponseData : RobotLibraryRecvDataFB;
  /// Timestamp
  Timestamp    : SystemTime;  
END_VAR
// Create log entry for Parameter start
CreateLogMessage      ( Timestamp   := Timestamp,
                        MessageType := MessageType.CMD,
                        Severity    := Severity.DEBUG,
                        MessageCode := 0,
                        MessageText := 'Parsed the following parameter(s) from response data:');
                        
// Create log entry for InvocationCounter
CreateLogMessagePara1 ( Timestamp   := Timestamp,
                        MessageType := MessageType.CMD,
                        Severity    := Severity.DEBUG,
                        MessageCode := 0,
                        MessageText := 'Response.InvocationCounter = {1}',
                        Para1       :=  USINT_TO_STRING(_response.InvocationCounter));

// Create log entry for Reserve
CreateLogMessagePara1 ( Timestamp   := Timestamp,
                        MessageType := MessageType.CMD,
                        Severity    := Severity.DEBUG,
                        MessageCode := 0,
                        MessageText := 'Response.Reserve = {1}',
                        Para1       :=  SINT_TO_STRING(_response.Reserved));

// Create log entry for OriginID
CreateLogMessagePara1 ( Timestamp   := Timestamp,
                        MessageType := MessageType.CMD,
                        Severity    := Severity.DEBUG,
                        MessageCode := 0,
                        MessageText := 'Response.OriginID = {1}',
                        Para1       :=  INT_TO_STRING(_response.OriginID));

// Create log entry for ForceStatus
CreateLogMessagePara1 ( Timestamp   := Timestamp,
                        MessageType := MessageType.CMD,
                        Severity    := Severity.DEBUG,
                        MessageCode := 0,
                        MessageText := 'Response.ForceStatus = {1}',
                        Para1       :=  BYTE_TO_STRING(_response.ForceStatus));
END_METHOD

METHOD PROTECTED Reset : DINT
VAR_INPUT
END_VAR
Reset := SUPER^.Reset();

Valid              := FALSE;
Busy               := FALSE;
CommandBuffered    := FALSE;
ParameterAccepted  := FALSE;
END_METHOD

END_FUNCTION_BLOCK

// Library/POUs/ForceControl/MC_ReadActualForce/MC_ReadActualForceFB
/// Read actual force/torque at TCP
FUNCTION_BLOCK MC_ReadActualForceFB EXTENDS RobotLibraryBaseExecuteFB
// ------------------------------------------------------------------------- 
//  SRCI Robot Library                                                
// ------------------------------------------------------------------------- 
//                                                                           
//  Object:      ReadActualForceFB                                       
//  Author:      Thorsten Brach                                                
//  Date:        2024-06-01
//
//  Description:                                              
//   
//                                                                           
//  Copyright: 
//    (C) 2024 Thorsten Brach. All rights reserved                                                                                                                                            
//             Licensed under the LGPL-3.0 license.
//                                                                           
//  Disclaimer:                                                                           
//    This project is provided without any guarantee and can be used for   
//    private and commercial purposes. Any use is at the user’s 
//    own risk and responsibility.
//
// -------------------------------------------------------------------------
VAR_INPUT
  /// Command parameter 
  ParCmd            : ReadActualForceParCmd;   
END_VAR

VAR_OUTPUT
  /// TRUE, while the following outputs return valid values:
  /// - ActualForce
  Valid             : BOOL;
  /// Command is transferred and confirmed by the RC
  CommandBuffered   : BOOL;
  /// Receiving of input parameter values has been acknowledged by RC
  ParameterAccepted : BOOL;
  /// Command output 
  OutCmd            : ReadActualForceOutCmd;        
END_VAR

VAR
  /// internal copy of command parameter 
 _parCmd            : ReadActualForceParCmd;
  /// command data to send
 _command           : ReadActualForceSendData;
  /// response data received
 _response          : ReadActualForceRecvData;      
END_VAR

SUPER^(AxesGroup := AxesGroup);

METHOD PROTECTED CheckFunctionSupported : BOOL
VAR_IN_OUT
  /// Robot assignment of function
  AxesGroup : AxesGroup; 
END_VAR
CheckFunctionSupported := AxesGroup.InternalData.RCSupportedFunctions.ReadActualForce;

IF ( NOT CheckFunctionSupported )
THEN
  // call base implementation for set error and create log entry
  SUPER^.CheckFunctionSupported(AxesGroup := AxesGroup);
END_IF
END_METHOD

METHOD PROTECTED CheckParameterChanged : BOOL
VAR_IN_OUT
  /// Robot assignment of function
  AxesGroup    : AxesGroup; 
END_VAR
// Check ParCmd Size is > 0, because MemCmp does not work correctly with size = 0
IF (SIZEOF(ParCmd) = 0) 
THEN 
  RETURN;
END_IF

// compare memory 
_parameterChanged := ( SysDepMemCmp(pData1 := ADR(ParCmd), pData2 := ADR(_parCmd), DataLen := SIZEOF(ParCmd)) <> RobotLibraryConstants.OK );

// check parameter valid ?
_parameterValid   := CheckParameterValid( AxesGroup := AxesGroup );

IF ((  _parameterChanged        )  AND 
    (  _parameterValid          )) OR
    (  _parameterUpdateInternal )  
THEN  
  // reset internal flag for send parameter update
 _parameterUpdateInternal := FALSE;
  // update internal copy of parameters 
 _parCmd := ParCmd;
  // inc parameter sequence
 _command.ParSeq := _command.ParSeq + 1;
  // update command data  
  CommandData := CreateCommandPayload(AxesGroup := AxesGroup); // ( Access via reference to rCommandFB in ACR )
  // notify active command register 
  AxesGroup.Acyclic.ActiveCommandRegister.NotifyParameterChanged := _uniqueID;
  // Reset parameter accepted flag
  ParameterAccepted := FALSE;  
END_IF
END_METHOD

METHOD INTERNAL CreateCommandPayload : RobotLibrarySendDataFB
VAR_IN_OUT
  /// Robot assignment of function
  AxesGroup : AxesGroup; 
END_VAR
// Table 6-733: Sent CMD payload (PLC to RC) of "ReadActualForce"
// --------------------------
// Header
// --------------------------
// Byte 00 : UINT       - Type HB     
// Byte 01 :            - Type LB    
// Byte 02 : USINT      - Reserve | ExecutionMode
// Byte 03 : USINT      - ParSeq  | Priority
// --------------------------
// Datablock
// --------------------------
// Byte 04 : SINT       - EmitterID[0]
// Byte 05 : SINT       - EmitterID[1]
// Byte 06 : SINT       - EmitterID[2]
// Byte 07 : SINT       - EmitterID[3]
// Byte 08 : SINT       - ListenerID
// Byte 09 : BYTE       - Reserved
// Byte 10 : USINT      - ToolNo
// Byte 11 : USINT      - FrameNo
// Byte 12 : USINT      - CalibrationData
// Byte 13 : USINT      - ReferenceType
// --------------------------
// set command parameter 
_command.CmdTyp          :=  CmdType.ReadActualForce;
_command.ExecMode        :=  ExecMode;
_command.ParSeq          := _command.ParSeq;
_command.Priority        :=  Priority;
_command.EmitterID[0]    := 0; {warning 'ToDo'}
_command.EmitterID[1]    := 0; {warning 'ToDo'}
_command.EmitterID[2]    := 0; {warning 'ToDo'}
_command.EmitterID[3]    := 0; {warning 'ToDo'}
_command.ListenerID      := _parCmd.ListenerID;
_command.Reserve         := 0;
_command.ToolNo          := _parCmd.ToolNo;
_command.FrameNo         := _parCmd.FrameNo;
_command.CalibrationData := _parCmd.CalibrationData;
_command.FrameNo         := _parCmd.FrameNo;
_command.ReferenceType   := _parCmd.ReferenceType;

// copy command data to header
_cmdHeader := _command;
// call base implementation to copy header to payload buffer
CreateCommandPayload := SUPER^.CreateCommandPayload(AxesGroup := AxesGroup);


// add command.EmitterID[0]
CreateCommandPayload.AddSint(_command.EmitterID[0]);
// add command.EmitterID[1]
CreateCommandPayload.AddSint(_command.EmitterID[1]);
// add command.EmitterID[2]
CreateCommandPayload.AddSint(_command.EmitterID[2]);
// add command.EmitterID[3]
CreateCommandPayload.AddSint(_command.EmitterID[3]);
// add command.ListenerID
CreateCommandPayload.AddSint(_command.ListenerID);
// add command.Reserve
CreateCommandPayload.AddByte(_command.Reserve);
// add command.ToolNo
CreateCommandPayload.AddUsint(_command.ToolNo);
// add command.FrameNo
CreateCommandPayload.AddUsint(_command.FrameNo);
// add command.CalibrationData
CreateCommandPayload.AddUsint(_command.CalibrationData);
// add command.ReferenceType
CreateCommandPayload.AddUsint(_command.ReferenceType);

// Create logging
CreateCommandPayloadLog(AxesGroup := AxesGroup);
END_METHOD

METHOD INTERNAL CreateCommandPayloadLog 
VAR_IN_OUT
  /// Robot assignment of function
  AxesGroup : AxesGroup; 
END_VAR
VAR 
  /// internal index for loops
 _idx : DINT;
END_VAR
// Create log entry for Parameter start
CreateLogMessage      ( Timestamp   := AxesGroup.InternalData.SystemTime,
                        MessageType := MessageType.CMD,
                        Severity    := Severity.DEBUG,
                        MessageCode := 0,
                        MessageText := 'Create command payload with the following parameter(s) :');

// Create log entry for EmitterID[x]
FOR _idx := 0 TO 3
DO
  CreateLogMessagePara2 ( Timestamp   := AxesGroup.InternalData.SystemTime,
                          MessageType := MessageType.CMD,
                          Severity    := Severity.DEBUG,
                          MessageCode := 0,
                          MessageText := 'Command.EmitterID[{2}] = {1}',
                          Para1       :=  SINT_TO_STRING(_command.EmitterID[_idx]),
                          Para2       :=  DINT_TO_STRING(_idx));
END_FOR

// Create log entry for ListenerID
CreateLogMessagePara1 ( Timestamp   := AxesGroup.InternalData.SystemTime,
                        MessageType := MessageType.CMD,
                        Severity    := Severity.DEBUG,
                        MessageCode := 0,
                        MessageText := 'Command.ListenerID = {1}',
                        Para1       :=  SINT_TO_STRING(_command.ListenerID));
                        
// Create log entry for Reserve
CreateLogMessagePara1 ( Timestamp   := AxesGroup.InternalData.SystemTime,
                        MessageType := MessageType.CMD,
                        Severity    := Severity.DEBUG,
                        MessageCode := 0,
                        MessageText := 'Command.Reserve = {1}',
                        Para1       :=  BYTE_TO_STRING(_command.Reserve));

// Create log entry for ToolNo
CreateLogMessagePara1 ( Timestamp   := AxesGroup.InternalData.SystemTime,
                        MessageType := MessageType.CMD,
                        Severity    := Severity.DEBUG,
                        MessageCode := 0,
                        MessageText := 'Command.ToolNo = {1}',
                        Para1       :=  USINT_TO_STRING(_command.ToolNo));
                        
// Create log entry for FrameNo
CreateLogMessagePara1 ( Timestamp   := AxesGroup.InternalData.SystemTime,
                        MessageType := MessageType.CMD,
                        Severity    := Severity.DEBUG,
                        MessageCode := 0,
                        MessageText := 'Command.FrameNo = {1}',
                        Para1       :=  USINT_TO_STRING(_command.FrameNo));
                                                
// Create log entry for CalibrationData
CreateLogMessagePara1 ( Timestamp   := AxesGroup.InternalData.SystemTime,
                        MessageType := MessageType.CMD,
                        Severity    := Severity.DEBUG,
                        MessageCode := 0,
                        MessageText := 'Command.CalibrationData = {1}',
                        Para1       :=  USINT_TO_STRING(_command.CalibrationData));

// Create log entry for ReferenceType
CreateLogMessagePara1 ( Timestamp   := AxesGroup.InternalData.SystemTime,
                        MessageType := MessageType.CMD,
                        Severity    := Severity.DEBUG,
                        MessageCode := 0,
                        MessageText := 'Command.ReferenceType = {1}',
                        Para1       :=  USINT_TO_STRING(_command.ReferenceType));
END_METHOD

METHOD FB_init : BOOL
VAR_INPUT
  /// if TRUE, the retain variables are initialized (warm start / cold start)
  bInitRetains : BOOL; 
  /// if TRUE, the instance afterwards gets moved into the copy code (online change)
  bInCopyCode  : BOOL;  
END_VAR
MyType := 'MC_ReadActualForceFB';

ExecMode := ExecutionMode.PARALLEL;
END_METHOD

METHOD PROTECTED OnCall
VAR_IN_OUT
  /// Robot assignment of function
  AxesGroup : AxesGroup; 
END_VAR
// call base implementation
SUPER^.OnCall(AxesGroup := AxesGroup);

CASE _stepCmd OF
  
  00:  IF ( _execute_R.Q )  
       THEN
         // Check function is supported and parameter are valid ?
         IF (( CheckFunctionSupported( AxesGroup := AxesGroup )) AND
             ( CheckParameterValid   ( AxesGroup := AxesGroup )))      
         THEN
           // set busy flag
           Busy := TRUE;
           // Reset command outputs
           SysDepMemSet(pDest := ADR(OutCmd), Value := 0, DataLen := SIZEOF(OutCmd));         
           // apply command parameter
          _parCmd := ParCmd;
           // init parameter sequence
          _command.ParSeq := 1;
           // create command data
           CommandData := CreateCommandPayload(AxesGroup := AxesGroup);
           // Add command to active command register
          _uniqueID := AxesGroup.Acyclic.ActiveCommandRegister.AddCmd( pCommandFB := ADR(THIS^ ));     
           // set timeout
           SetTimeout(PT := _timeoutCmd, rTimer := _timerCmd);
           // inc step counter
          _stepCmd := _stepCmd + 1;
         END_IF 
       END_IF
     

  01:  // Wait for responce received
       IF ( _responseReceived )
       THEN
         // reset response received flag
        _responseReceived := FALSE;

         CASE  _response.State 
         OF
           CmdMessageState.BUFFERED : CommandBuffered   := TRUE;
           CmdMessageState.ACTIVE   : ParameterAccepted := TRUE;
           CmdMessageState.Done     : Done              := TRUE;
           CmdMessageState.ERROR    : Error             := TRUE;
         END_CASE
                
         // Done, Aborted or Error ?
         IF (_response.State >= CmdMessageState.DONE )
         THEN
           // Reset Busy flag
           Busy := FALSE;
           // Update results
           OutCmd.OriginID          := _response.OriginID;
           OutCmd.InvocationCounter := _response.InvocationCounter;
           OutCmd.ActualForce       := _response.ActualForce;
           // set timeout
           SetTimeout(PT := _timeoutCmd, rTimer := _timerCmd);
           // inc step counter
          _stepCmd := _stepCmd + 1; 
         END_IF
       END_IF


  02: IF ( NOT Execute)
      THEN
        Reset();
      END_IF     

ELSE
  // invalid step
  ErrorID := RobotLibraryEvents.ERR_INVALID_STEP;
END_CASE


// Reset FB
IF ( NOT Execute )
THEN
  Reset();  
END_IF
END_METHOD

METHOD INTERNAL ParseResponsePayload : DINT
VAR_INPUT
  /// Response data
  ResponseData : RobotLibraryRecvDataFB;
  /// Timestamp
  Timestamp    : SystemTime;  
END_VAR
VAR 
  /// internal index for loops
 _idx : DINT;
END_VAR
// Table 6-734: Received CMD payload (RC to PLC) of "ReadActualForce"
// --------------------------
// Header
// --------------------------
// Byte 00 : USINT      - ParSeq | State     
// Byte 01 : SINT       - AlarmMessageSeverity    
// Byte 02 : UINT       - AlarmMessageCode HB
// Byte 03 :            - AlarmMessageCode LB
// --------------------------
// Datablock
// --------------------------
// Byte 04 : USINT      - InvocationCounter
// Byte 05 : SINT       - Reserved
// Byte 06 : INT        - OriginID LW HB
// Byte 07 :            - OriginID LW LB
// Byte 08 : REAL       - ActualForce[0] HW HB
// Byte 09 :            - ActualForce[0] HW LB
// Byte 10 :            - ActualForce[0] LW HB
// Byte 11 :            - ActualForce[0] LW LB
// Byte 12 : REAL       - ActualForce[1] HW HB
// Byte 13 :            - ActualForce[1] HW LB
// Byte 24 :            - ActualForce[1] LW HB
// Byte 15 :            - ActualForce[1] LW LB
// Byte 16 : REAL       - ActualForce[2] HW HB
// Byte 17 :            - ActualForce[2] HW LB
// Byte 18 :            - ActualForce[2] LW HB
// Byte 19 :            - ActualForce[2] LW LB
// Byte 20 : REAL       - ActualForce[3] HW HB
// Byte 21 :            - ActualForce[3] HW LB
// Byte 22 :            - ActualForce[3] LW HB
// Byte 23 :            - ActualForce[3] LW LB
// Byte 24 : REAL       - ActualForce[4] HW HB
// Byte 25 :            - ActualForce[4] HW LB
// Byte 26 :            - ActualForce[4] LW HB
// Byte 27 :            - ActualForce[4] LW LB
// Byte 28 : REAL       - ActualForce[5] HW HB
// Byte 29 :            - ActualForce[5] HW LB
// Byte 30 :            - ActualForce[5] LW HB
// Byte 31 :            - ActualForce[5] LW LB
// --------------------------
// call base implementation to parse the header from payload buffer
ResponseData.PayloadPtr := SUPER^.ParseResponsePayload(ResponseData := ResponseData, Timestamp := Timestamp);

// copy parsed header to response
_response.ParSeq                := _rspHeader.ParSeq;
_response.State                 := _rspHeader.State;
_response.AlarmMessageSeverity  := _rspHeader.AlarmMessageSeverity;
_response.AlarmMessageCode      := _rspHeader.AlarmMessageCode;

// Get Response.InvocationCounter
_response.InvocationCounter := ResponseData.GetUsint();
// Get Response.Reserved
_response.Reserved := ResponseData.GetSint();
// Get Response.InvocationCounter
_response.OriginID := ResponseData.GetInt();

FOR _idx := 0 TO 5
DO
  // Get Response.ActualForce[x]
 _response.ActualForce[_idx] := ResponseData.GetReal();
END_FOR

// Create logging
ParseResponsePayloadLog(ResponseData := ResponseData, Timestamp := Timestamp);
END_METHOD

METHOD INTERNAL ParseResponsePayloadLog
VAR_INPUT
  /// Response data
  ResponseData : RobotLibraryRecvDataFB;
  /// Timestamp
  Timestamp    : SystemTime;  
END_VAR
VAR 
  /// internal index for loops
 _idx : DINT;
END_VAR
// Create log entry for Parameter start
CreateLogMessage      ( Timestamp   := Timestamp,
                        MessageType := MessageType.CMD,
                        Severity    := Severity.DEBUG,
                        MessageCode := 0,
                        MessageText := 'Parsed the following parameter(s) from response data:');
                        
// Create log entry for InvocationCounter
CreateLogMessagePara1 ( Timestamp   := Timestamp,
                        MessageType := MessageType.CMD,
                        Severity    := Severity.DEBUG,
                        MessageCode := 0,
                        MessageText := 'Response.InvocationCounter = {1}',
                        Para1       :=  USINT_TO_STRING(_response.InvocationCounter));

// Create log entry for Reserve
CreateLogMessagePara1 ( Timestamp   := Timestamp,
                        MessageType := MessageType.CMD,
                        Severity    := Severity.DEBUG,
                        MessageCode := 0,
                        MessageText := 'Response.Reserve = {1}',
                        Para1       :=  SINT_TO_STRING(_response.Reserved));

// Create log entry for OriginID
CreateLogMessagePara1 ( Timestamp   := Timestamp,
                        MessageType := MessageType.CMD,
                        Severity    := Severity.DEBUG,
                        MessageCode := 0,
                        MessageText := 'Response.OriginID = {1}',
                        Para1       :=  INT_TO_STRING(_response.OriginID));

// Create log entry for ActualForce[x]
FOR _idx := 0 TO 5
DO
  CreateLogMessagePara2 ( Timestamp   := Timestamp,
                          MessageType := MessageType.CMD,
                          Severity    := Severity.DEBUG,
                          MessageCode := 0,
                          MessageText := 'Response.ActualForce[{2}] = {1}',
                          Para1       :=  REAL_TO_STRING(_response.ActualForce[_idx]),
                          Para2       :=  DINT_TO_STRING(_idx));
END_FOR
END_METHOD

METHOD PROTECTED Reset : DINT
VAR_INPUT
END_VAR
Reset := SUPER^.Reset();

Done               := FALSE;
Busy               := FALSE;
Valid              := FALSE;
ParameterAccepted  := FALSE;
CommandBuffered    := FALSE;
END_METHOD

END_FUNCTION_BLOCK

// Library/POUs/General/MC_CreateServerLog_ToDo/MC_CreateServerLog_ToDo
FUNCTION_BLOCK MC_CreateServerLog_ToDo EXTENDS RobotLibraryBaseFB
VAR
END_VAR

METHOD FB_init : BOOL
VAR_INPUT
  /// if TRUE, the retain variables are initialized (warm start / cold start)
  bInitRetains : BOOL; 
  /// if TRUE, the instance afterwards gets moved into the copy code (online change)
  bInCopyCode  : BOOL;  
END_VAR
MyType := 'MC_CreateServerLogFB';
END_METHOD

END_FUNCTION_BLOCK

// Library/POUs/General/MC_EnableRobot/MC_EnableRobotFB
/// Enable/Disable robot into RA power state "Enabled"
FUNCTION_BLOCK MC_EnableRobotFB EXTENDS RobotLibraryBaseEnableFB
// ------------------------------------------------------------------------- 
//  SRCI Robot Library                                                
// ------------------------------------------------------------------------- 
//                                                                           
//  Object:      EnableRobotFB                                       
//  Author:      Thorsten Brach                                                
//  Date:        2024-06-01
//
//  Description:                                              
//   
//                                                                           
//  Copyright: 
//    (C) 2024 Thorsten Brach. All rights reserved                                                                                                                                            
//             Licensed under the LGPL-3.0 license.
//                                                                           
//  Disclaimer:                                                                           
//    This project is provided without any guarantee and can be used for   
//    private and commercial purposes. Any use is at the user’s 
//    own risk and responsibility.
//
// -------------------------------------------------------------------------
VAR_INPUT
  /// Command parameter 
  ParCmd            : EnableRobotParCmd;
END_VAR


VAR_OUTPUT
  /// Command is transferred and confirmed by the RC
  CommandBuffered   : BOOL;
  /// Receiving of input parameter values has been acknowledged by RC
  ParameterAccepted : BOOL;
  /// command results
  OutCmd            : EnableRobotOutCmd;
END_VAR

VAR
  /// internal copy of command parameter 
 _parCmd            : EnableRobotParCmd;
  /// command data to send
 _command           : EnableRobotSendData;
  /// response data received
 _response          : EnableRobotRecvData;
END_VAR

SUPER^(AxesGroup := AxesGroup);

METHOD PROTECTED CheckFunctionSupported : BOOL
VAR_IN_OUT
  /// Robot assignment of function
  AxesGroup : AxesGroup; 
END_VAR
CheckFunctionSupported := AxesGroup.InternalData.RCSupportedFunctions.EnableRobot;

IF ( NOT CheckFunctionSupported )
THEN
  // call base implementation for set error and create log entry
  SUPER^.CheckFunctionSupported(AxesGroup := AxesGroup);
END_IF
END_METHOD

METHOD PROTECTED CheckParameterChanged : BOOL
VAR_IN_OUT
  /// Robot assignment of function
  AxesGroup    : AxesGroup; 
END_VAR
// Check ParCmd Size is > 0, because MemCmp does not work correctly with size = 0
IF (SIZEOF(ParCmd) = 0) 
THEN 
  RETURN;
END_IF

// compare memory 
_parameterChanged := ( SysDepMemCmp(pData1 := ADR(ParCmd), pData2 := ADR(_parCmd), DataLen := SIZEOF(ParCmd)) <> RobotLibraryConstants.OK );

// check parameter valid ?
_parameterValid   := CheckParameterValid( AxesGroup := AxesGroup );

IF ((  _parameterChanged        )  AND 
    (  _parameterValid          )) OR
    (  _parameterUpdateInternal )  
THEN  
  // reset internal flag for send parameter update
 _parameterUpdateInternal := FALSE;
  // update internal copy of parameters 
 _parCmd := ParCmd;
  // inc parameter sequence
 _command.ParSeq := _command.ParSeq + 1;
  // update command data  
  CommandData := CreateCommandPayload(AxesGroup := AxesGroup); // ( Access via reference to rCommandFB in ACR )
  // notify active command register 
  AxesGroup.Acyclic.ActiveCommandRegister.NotifyParameterChanged := _uniqueID;
  // Reset parameter accepted flag
  ParameterAccepted := FALSE;  
END_IF
END_METHOD

METHOD INTERNAL CreateCommandPayload : RobotLibrarySendDataFB
VAR_IN_OUT
  /// Robot assignment of function
  AxesGroup : AxesGroup; 
END_VAR
// Table 6-25: Sent CMD payload (PLC to RC) of "EnableRobot"
// --------------------------
// Header
// --------------------------
// Byte 00 : UINT  - Type HB     
// Byte 01 :       - Type LB    
// Byte 02 : USINT - Reserve | ExecutionMode
// Byte 03 : USINT - ParSeq  | Priority
// --------------------------
// Datablock
// --------------------------
// Byte 04 : BOOL  - Enable
// Byte 05 : BOOL  - HoldToRun
// Byte 06 : USINT - StepMode   
// Byte 07 : BOOL  - ManualStep
// --------------------------
// set command parameter 
_command.CmdTyp    :=  CmdType.EnableRobot;
_command.ExecMode  :=  ExecMode;
_command.ParSeq    := _command.ParSeq;
_command.Priority  :=  Priority;
_command.Enable    :=  Enable;
_command.HoldToRun := _parCmd.HoldToRun;
_command.StepMode  := _parCmd.StepMode;
_command.ManualStep:= _parCmd.ManualStep;


// copy command data to header
_cmdHeader := _command;
// call base implementation to copy header to payload buffer
CreateCommandPayload := SUPER^.CreateCommandPayload(AxesGroup := AxesGroup);

// add command.Enable
CreateCommandPayload.AddBool(_command.Enable);
// add command.StepMode
CreateCommandPayload.AddUsint(_command.StepMode);
// add command.HoldToRun
CreateCommandPayload.AddBool(_command.HoldToRun);
// add command.ManualStep
CreateCommandPayload.AddBool(_command.ManualStep);                      

// Create logging
CreateCommandPayloadLog(AxesGroup := AxesGroup);
END_METHOD

METHOD INTERNAL CreateCommandPayloadLog 
VAR_IN_OUT
  /// Robot assignment of function
  AxesGroup : AxesGroup; 
END_VAR
// Create log entry for Parameter start
CreateLogMessage      ( Timestamp   := AxesGroup.InternalData.SystemTime,
                        MessageType := MessageType.CMD,
                        Severity    := Severity.DEBUG,
                        MessageCode := 0,
                        MessageText := 'Create command payload with the following parameter(s) :');

// Create log entry for Enable
CreateLogMessagePara1 ( Timestamp   := AxesGroup.InternalData.SystemTime,
                        MessageType := MessageType.CMD,
                        Severity    := Severity.DEBUG,
                        MessageCode := 0,
                        MessageText := 'Command.Enable = {1}',
                        Para1       :=  BOOL_TO_STRING(_command.Enable));

// Create log entry for HoldToRun
CreateLogMessagePara1 ( Timestamp   := AxesGroup.InternalData.SystemTime,
                        MessageType := MessageType.CMD,
                        Severity    := Severity.DEBUG,
                        MessageCode := 0,
                        MessageText := 'Command.HoldToRun = {1}',
                        Para1       :=  BOOL_TO_STRING(_command.HoldToRun));
                        
// Create log entry for StepMode
CreateLogMessagePara1 ( Timestamp   := AxesGroup.InternalData.SystemTime,
                        MessageType := MessageType.CMD,
                        Severity    := Severity.DEBUG,
                        MessageCode := 0,
                        MessageText := 'Command.StepMode = {1}',
                        Para1       :=  USINT_TO_STRING(_command.StepMode));
                                                
// Create log entry for ManualStep
CreateLogMessagePara1 ( Timestamp   := AxesGroup.InternalData.SystemTime,
                        MessageType := MessageType.CMD,
                        Severity    := Severity.DEBUG,
                        MessageCode := 0,
                        MessageText := 'Command.ManualStep = {1}',
                        Para1       :=  BOOL_TO_STRING(_command.ManualStep));
END_METHOD

METHOD FB_init : BOOL
VAR_INPUT
  /// if TRUE, the retain variables are initialized (warm start / cold start)
  bInitRetains : BOOL; 
  /// if TRUE, the instance afterwards gets moved into the copy code (online change)
  bInCopyCode  : BOOL;  
END_VAR
MyType := 'MC_EnableRobotFB';
ExecMode := ExecutionMode.PARALLEL;
END_METHOD

METHOD PROTECTED OnCall
VAR_IN_OUT
  /// Robot assignment of function
  AxesGroup : AxesGroup; 
END_VAR
SUPER^.OnCall(AxesGroup := AxesGroup);

CASE _stepCmd OF
  
  00:  IF ( _enable_R.Q ) 
       THEN
         // reset the rising edge
        _enable_R();       
         // reset the falling edge
        _enable_F();      

         // Check function is supported and parameter are valid ?
         IF (( CheckFunctionSupported( AxesGroup := AxesGroup )) AND
             ( CheckParameterValid   ( AxesGroup := AxesGroup )))      
         THEN
           // set busy flag
           Busy := TRUE;
           // Reset command outputs
           SysDepMemSet(pDest := ADR(OutCmd), Value := 0, DataLen := SIZEOF(OutCmd));         
           // apply command parameter
          _parCmd := ParCmd;
           // init parameter sequence
          _command.ParSeq := 1;
           // create command data
           CommandData := CreateCommandPayload(AxesGroup := AxesGroup);
           // Add command to active command register
          _uniqueID := AxesGroup.Acyclic.ActiveCommandRegister.AddCmd( pCommandFB := ADR(THIS^ ));     
           // set timeout
           SetTimeout(PT := _timeoutCmd, rTimer := _timerCmd);
           // inc step counter
          _stepCmd := _stepCmd + 1; 
         END_IF
       END_IF
     

  01:  // Wait for responce received
       IF ( _responseReceived )
       THEN
         // reset response received flag
        _responseReceived := FALSE;

         CASE  _response.State 
         OF
           CmdMessageState.BUFFERED    : CommandBuffered    := TRUE;
           CmdMessageState.ACTIVE      : ParameterAccepted  := TRUE;           
           CmdMessageState.ERROR       : Error              := TRUE;
         END_CASE
         
         // Update results
         Enabled := _response.Enabled;
                
         // Done, Aborted or Error ?
         IF (_response.State >= CmdMessageState.DONE )
         THEN
           // reset busy flag
           Enabled := FALSE;          
           // Delete command from active command register, if not yet happend
           AxesGroup.Acyclic.ActiveCommandRegister.RemoveCmd( UniqueID := _uniqueID); 
           // set timeout
           SetTimeout(PT := _timeoutCmd, rTimer := _timerCmd);
           // inc step counter
          _stepCmd := _stepCmd + 1; 
         END_IF
       END_IF
       
       // do not abort directly, so that the ParSeq update can be send
       IF ( _enable_R.Q ) OR ( _enable_F.Q ) 
       THEN
         // trigger parameter update to disable Enable
        _parameterUpdateInternal := TRUE;
         // reset the rising edge
        _enable_R();       
         // reset the falling edge
        _enable_F();       
       END_IF


  02:  IF (NOT Enable)
       THEN
         Reset();  
       END_IF

ELSE
  // invalid step
  ErrorID := RobotLibraryEvents.ERR_INVALID_STEP;
END_CASE



// Reset FB
IF (( _enable_R.Q ) OR
    ( _enable_F.Q ))
THEN
  Reset();
END_IF
END_METHOD

METHOD INTERNAL ParseResponsePayload : DINT
VAR_INPUT
  /// Response data
  ResponseData : RobotLibraryRecvDataFB;
  /// Timestamp
  Timestamp    : SystemTime;  
END_VAR
// Table 6-26: Received CMD payload (RC to PLC) of "EnableRobot"
// --------------------------
// Header
// --------------------------
// Byte 00 : USINT - ParSeq | State     
// Byte 01 : SINT  - AlarmMessageSeverity    
// Byte 02 : UINT  - AlarmMessageCode HB
// Byte 03 :       - AlarmMessageCode LB
// --------------------------
// Datablock
// --------------------------
// Byte 04 : BOOL  - Enabled
// --------------------------
// call base implementation to parse the header from payload buffer
ResponseData.PayloadPtr := SUPER^.ParseResponsePayload(ResponseData := ResponseData, Timestamp := Timestamp);

// copy parsed header to response
_response.ParSeq               := _rspHeader.ParSeq;
_response.State                := _rspHeader.State;
_response.AlarmMessageSeverity := _rspHeader.AlarmMessageSeverity;
_response.AlarmMessageCode     := _rspHeader.AlarmMessageCode;

// Get Response.Enabled
_response.Enabled := ResponseData.GetBool();

// Create logging
ParseResponsePayloadLog(ResponseData := ResponseData, Timestamp := Timestamp);
END_METHOD

METHOD INTERNAL ParseResponsePayloadLog
VAR_INPUT
  /// Response data
  ResponseData : RobotLibraryRecvDataFB;
  /// Timestamp
  Timestamp    : SystemTime;  
END_VAR
// Create log entry for Parameter start
CreateLogMessage      ( Timestamp   := Timestamp,
                        MessageType := MessageType.CMD,
                        Severity    := Severity.DEBUG,
                        MessageCode := 0,
                        MessageText := 'Parsed the following parameter(s) from response data:');
                        
// Create log entry for Enabled
CreateLogMessagePara1 ( Timestamp   := Timestamp,
                        MessageType := MessageType.CMD,
                        Severity    := Severity.DEBUG,
                        MessageCode := 0,
                        MessageText := 'Response.Enabled = {1}',
                        Para1       :=  BOOL_TO_STRING(_response.Enabled));
END_METHOD

METHOD PROTECTED Reset : DINT
VAR_INPUT
END_VAR
SUPER^.Reset();

Busy               := FALSE;
CommandBuffered    := FALSE;
ParameterAccepted  := FALSE;
END_METHOD

END_FUNCTION_BLOCK

// Library/POUs/General/MC_GroupReset/MC_GroupResetFB
/// Acknowledgement all pending errors
FUNCTION_BLOCK MC_GroupResetFB EXTENDS RobotLibraryBaseExecuteFB
// ------------------------------------------------------------------------- 
//  SRCI Robot Library                                                
// ------------------------------------------------------------------------- 
//                                                                           
//  Object:      GroupResetFB                                       
//  Author:      Thorsten Brach                                                
//  Date:        2024-06-01
//
//  Description:                                              
//   
//                                                                           
//  Copyright: 
//    (C) 2024 Thorsten Brach. All rights reserved                                                                                                                                            
//             Licensed under the LGPL-3.0 license.
//                                                                           
//  Disclaimer:                                                                           
//    This project is provided without any guarantee and can be used for   
//    private and commercial purposes. Any use is at the user’s 
//    own risk and responsibility.
//
// -------------------------------------------------------------------------
VAR_INPUT
  /// Command parameter 
  ParCmd          : GroupResetParCmd;      
END_VAR

VAR_OUTPUT
  /// Command output 
  OutCmd          : GroupResetOutCmd;   
  /// Command is transferred and confirmed by the RC
  CommandBuffered : BOOL;     
END_VAR
VAR
  /// internal copy of command parameter 
 _parCmd          : GroupResetParCmd;
  /// command data to send
 _command         : GroupResetSendData;
  /// response data received
 _response        : GroupResetRecvData;      
END_VAR

SUPER^(AxesGroup := AxesGroup);

METHOD PROTECTED CheckFunctionSupported : BOOL
VAR_IN_OUT
  /// Robot assignment of function
  AxesGroup : AxesGroup; 
END_VAR
CheckFunctionSupported := AxesGroup.InternalData.RCSupportedFunctions.GroupReset;

IF ( NOT CheckFunctionSupported )
THEN
  // call base implementation for set error and create log entry
  SUPER^.CheckFunctionSupported(AxesGroup := AxesGroup);
END_IF
END_METHOD

METHOD PROTECTED CheckParameterChanged : BOOL
VAR_IN_OUT
  /// Robot assignment of function
  AxesGroup    : AxesGroup; 
END_VAR
IF (SIZEOF(ParCmd) = 0)
THEN
  RETURN;
END_IF
 
// compare memory
_parameterChanged := ( SysDepMemCmp(pData1 := ADR(ParCmd), pData2 := ADR(_parCmd), DataLen := SIZEOF(ParCmd)) <> RobotLibraryConstants.OK );

// check parameter valid ?
_parameterValid   := CheckParameterValid( AxesGroup := AxesGroup );

IF ((  _parameterChanged        )  AND 
    (  _parameterValid          )) OR
    (  _parameterUpdateInternal )  
THEN  
  // reset internal flag for send parameter update
 _parameterUpdateInternal := FALSE;
  // update internal copy of parameters 
 _parCmd := ParCmd;
  // inc parameter sequence
 _command.ParSeq := _command.ParSeq + 1;
  // update command data  
  CommandData := CreateCommandPayload(AxesGroup := AxesGroup); // ( Access via reference to rCommandFB in ACR )
  // notify active command register 
  AxesGroup.Acyclic.ActiveCommandRegister.NotifyParameterChanged := _uniqueID;
END_IF
END_METHOD

METHOD INTERNAL CreateCommandPayload : RobotLibrarySendDataFB
VAR_IN_OUT
  /// Robot assignment of function
  AxesGroup : AxesGroup; 
END_VAR
// Table 6-31: Sent CMD payload (PLC to RC) of "GroupReset"
// --------------------------
// Header
// --------------------------
// Byte 00 : UINT  - Type HB     
// Byte 01 :       - Type LB    
// Byte 02 : USINT - Reserve | ExecutionMode
// Byte 03 : USINT - ParSeq  | Priority
// --------------------------
// set command parameter 
_command.CmdTyp     :=  CmdType.GroupReset;
_command.ExecMode   :=  ExecMode;
_command.ParSeq     := _command.ParSeq;
_command.Priority   :=  Priority;


// copy command data to header
_cmdHeader := _command;
// call base implementation to copy header to payload buffer
CreateCommandPayload := SUPER^.CreateCommandPayload(AxesGroup := AxesGroup);

// Create logging
CreateCommandPayloadLog(AxesGroup := AxesGroup);
END_METHOD

METHOD INTERNAL CreateCommandPayloadLog
VAR_IN_OUT
  /// Robot assignment of function
  AxesGroup : AxesGroup; 
END_VAR
// Create log entry for Parameter start
CreateLogMessage      ( Timestamp   := AxesGroup.InternalData.SystemTime,
                        MessageType := MessageType.CMD,
                        Severity    := Severity.DEBUG,
                        MessageCode := 0,
                        MessageText := 'Create command payload without additional parameter(s)');
END_METHOD

METHOD FB_init : BOOL
VAR_INPUT
  /// if TRUE, the retain variables are initialized (warm start / cold start)
  bInitRetains : BOOL; 
  /// if TRUE, the instance afterwards gets moved into the copy code (online change)
  bInCopyCode  : BOOL;  
END_VAR
MyType := 'MC_GroupResetFB';

ExecMode := ExecutionMode.PARALLEL;
END_METHOD

METHOD PROTECTED OnCall
VAR_IN_OUT
  /// Robot assignment of function
  AxesGroup : AxesGroup; 
END_VAR
// call base implementation
SUPER^.OnCall(AxesGroup := AxesGroup);

CASE _stepCmd OF
  
  00:  IF ( _execute_R.Q )
       THEN
         IF (( CheckFunctionSupported( AxesGroup := AxesGroup )) AND
             ( CheckParameterValid   ( AxesGroup := AxesGroup )))      
         THEN
           // set busy flag
           Busy := TRUE;
           // Reset command outputs
           SysDepMemSet(pDest := ADR(OutCmd), Value := 0, DataLen := SIZEOF(OutCmd));         
           // apply command parameter
          _parCmd := ParCmd;
           // init parameter sequence
          _command.ParSeq := 1;
           // create command data
           CommandData := CreateCommandPayload(AxesGroup := AxesGroup);
           // Add command to active command register
          _uniqueID := AxesGroup.Acyclic.ActiveCommandRegister.AddCmd( pCommandFB := ADR(THIS^ ));     
           // set timeout
           SetTimeout(PT := _timeoutCmd, rTimer := _timerCmd);
           // inc step counter
          _stepCmd := _stepCmd + 1;
         END_IF 
       END_IF
     

  01:  // Wait for responce received
       IF ( _responseReceived )
       THEN
         // reset response received flag
        _responseReceived := FALSE;

